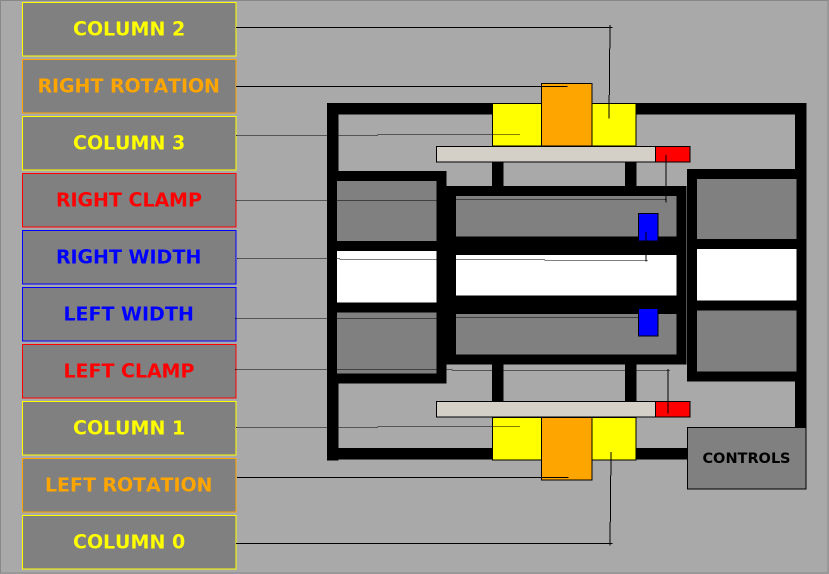
VISUALIZATION machineMapScreen  // 829x574
    Group (327,83 479x406)
        Rectangle (165,20 11x357)
        Rectangle (298,20 11x357)
        Rectangle (119,103 240x60)
        Rectangle (119,221 240x60)
        Rectangle (1,20 478x11)
        Rectangle (0,365 478x11)
        Rectangle (0,20 11x357)
        Rectangle (468,20 11x357)
        Rectangle (0,88 119x89)
        Rectangle (0,211 119x89)
        Rectangle (0,158 119x71)
        Rectangle (360,86 119x89)
        Rectangle (360,209 119x89)
        Rectangle (360,156 119x71)
        Rectangle (119,162 240x60)
        Rectangle (360,344 119x62), "CONTROLS"
        Rectangle (165,20 51x43)
        Rectangle (258,20 51x43)
        Rectangle (214,0 51x63)
        Rectangle (109,63 231x16)
        Rectangle (328,63 35x16)
        Rectangle (165,334 51x43)
        Rectangle (258,334 51x43)
        Rectangle (214,334 51x63)
        Rectangle (109,318 231x16)
        Rectangle (328,318 35x16)
    Rectangle (22,2 214x54), "COLUMN 2"
    Rectangle (22,59 214x54), "RIGHT ROTATION"
    Rectangle (22,116 214x54), "COLUMN 3"
    Rectangle (22,173 214x54), "RIGHT CLAMP"
    Rectangle (22,230 214x54), "RIGHT WIDTH"
    Rectangle (22,287 214x54), "LEFT WIDTH"
    Rectangle (22,344 214x54), "LEFT CLAMP"
    Rectangle (22,401 214x54), "COLUMN 1"
    Rectangle (22,515 214x54), "COLUMN 0"
    Rectangle (22,458 214x54), "LEFT ROTATION"
    Line (236,27) (612,27)
    Line (609,118) (610,25)
    Line (236,86) (567,86)
    Line (236,135) (519,134)
    Line (236,200) (665,199)
    Line (237,258) (647,260)
    Line (235,318) (640,317)
    Line (235,369) (669,370)
    Rectangle (638,213 20x28)
    Rectangle (638,308 20x28)
    Line (666,202) (666,155)
    Line (646,261) (646,232)
    Line (668,413) (668,369)
    Line (236,427) (519,426)
    Line (236,543) (612,543)
    Line (610,545) (611,452)
    Line (237,477) (568,477)
END_VISUALIZATION

(* stored: Version 1.1.0.1, ProductVersion 3.1.4024.13
   Visu machineMapScreen: Id {38e19128-55c1-4aa5-9ab6-0d4856cb7fe6} *)
